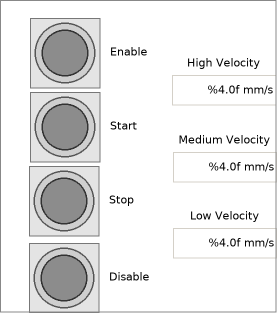
VISUALIZATION Controls  // 277x313
    PushSwitchLed (30,18 70x70), variable: MAIN.MainCommands.Enable, behaviour: TOGGLE, style: Switch-PushSwitchLed-Gray
    Label (107,37 75x30), "Enable"
    Label (107,111 75x30), "Start"
    PushSwitchLed (30,92 70x70), variable: MAIN.MainCommands.Start, behaviour: TOGGLE, style: Switch-PushSwitchLed-Gray
    Label (106,185 75x30), "Stop"
    PushSwitchLed (29,166 70x70), variable: MAIN.MainCommands.Stop, behaviour: TOGGLE, style: Switch-PushSwitchLed-Gray
    Label (106,262 75x30), "Disable"
    PushSwitchLed (29,243 70x70), variable: MAIN.MainCommands.Disable, behaviour: TOGGLE, style: Switch-PushSwitchLed-Gray
    Textfield (172,75 104x30), "%4.0f mm/s", text variable: MAIN.highVelocity
        OnMouseClick: write the text variable via VisuDialogs.Numpad, min 1, max 2000, format %f.0
    Label (175,54 97x18), "High Velocity"
    Textfield (173,152 104x30), "%4.0f mm/s", text variable: MAIN.mediumVelocity
        OnMouseClick: write the text variable via VisuDialogs.Numpad, min 1, max 2000, format %f.0
    Label (176,131 97x18), "Medium Velocity"
    Textfield (173,228 104x30), "%4.0f mm/s", text variable: MAIN.lowVelocity
        OnMouseClick: write the text variable via VisuDialogs.Numpad, min 1, max 2000, format %f.0
    Label (176,207 97x18), "Low Velocity"
END_VISUALIZATION

(* stored: Version 1.1.0.1, ProductVersion 3.1.4026.8
   Visu Controls: Id {d671d5e2-5681-0862-25f9-9de6f25977db} *)
